// SIMATIC S7-200 project (STEP 7-Micro/WIN), CPU 224XP REL 02.01

SYMBOL_TABLE USUARIO1
P_DERECHA        I0.0
P_IZQUIERDA      I0.1
P_PARO           I0.2
R_TERMICO        I0.3
M_DERECHA        Q0.0
LED_DERECHA      Q0.1
M_IZQUIERDA      Q0.2
LED_IZQUIERDA    Q0.3
LED_PARO         Q0.4
LED_TERMICO      Q0.5
END_SYMBOL_TABLE

SYMBOL_TABLE Símbolos S7-200
Primer_ciclo_ON  SM0.1    // ON sólo en el primer ciclo
END_SYMBOL_TABLE

ORGANIZATION_BLOCK PRINCIPAL:OB1
TITLE=COMENTARIOS DEL PROGRAMA
BEGIN
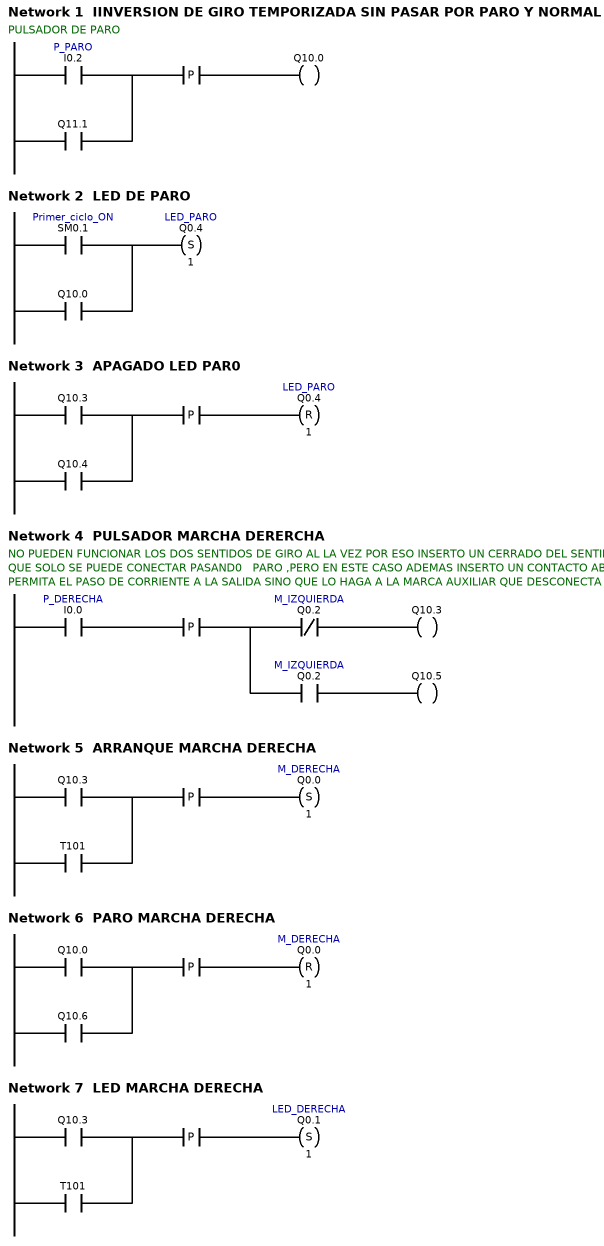
Network 1 // IINVERSION DE GIRO TEMPORIZADA SIN PASAR POR PARO Y NORMAL PASANDO POR PARO
// PULSADOR DE PARO
LD     P_PARO:I0.2
O      Q11.1
EU
=      Q10.0
Network 2 // LED DE PARO
LD     Primer_ciclo_ON:SM0.1
O      Q10.0
S      LED_PARO:Q0.4, 1
Network 3 // APAGADO LED PAR0
LD     Q10.3
O      Q10.4
EU
R      LED_PARO:Q0.4, 1
Network 4 // PULSADOR MARCHA DERERCHA
// NO PUEDEN FUNCIONAR LOS DOS SENTIDOS DE GIRO AL LA VEZ POR ESO INSERTO UN CERRADO DEL SENTIDO CONTRARIO ANTES DE LA MARCA QUE ME CONECTA AMBOS SENTIDOS DE TAL FORMA QUE SOLO SE PUEDE CONECTAR PASAND0   PARO ,PERO EN ESTE CASO ADEMAS INSERTO UN CONTACTO ABIERTO QUE CONECTA OTRA MARCA,CUAMDO YO PRESIONE EL SENTIDO QUE ELIJA NO ME PERMITA EL PASO DE CORRIENTE A LA SALIDA SINO QUE LO HAGA A LA MARCA AUXILIAR QUE DESCONECTA EL SENTIDO CONTRARIO Y TEMPORIZA PARA CONECTAR EL ELEGIDO.
LD     P_DERECHA:I0.0
EU
LPS
AN     M_IZQUIERDA:Q0.2
=      Q10.3
LPP
A      M_IZQUIERDA:Q0.2
=      Q10.5
Network 5 // ARRANQUE MARCHA DERECHA
LD     Q10.3
O      T101
EU
S      M_DERECHA:Q0.0, 1
Network 6 // PARO MARCHA DERECHA

LD     Q10.0
O      Q10.6
EU
R      M_DERECHA:Q0.0, 1
Network 7 // LED MARCHA DERECHA
LD     Q10.3
O      T101
EU
S      LED_DERECHA:Q0.1, 1
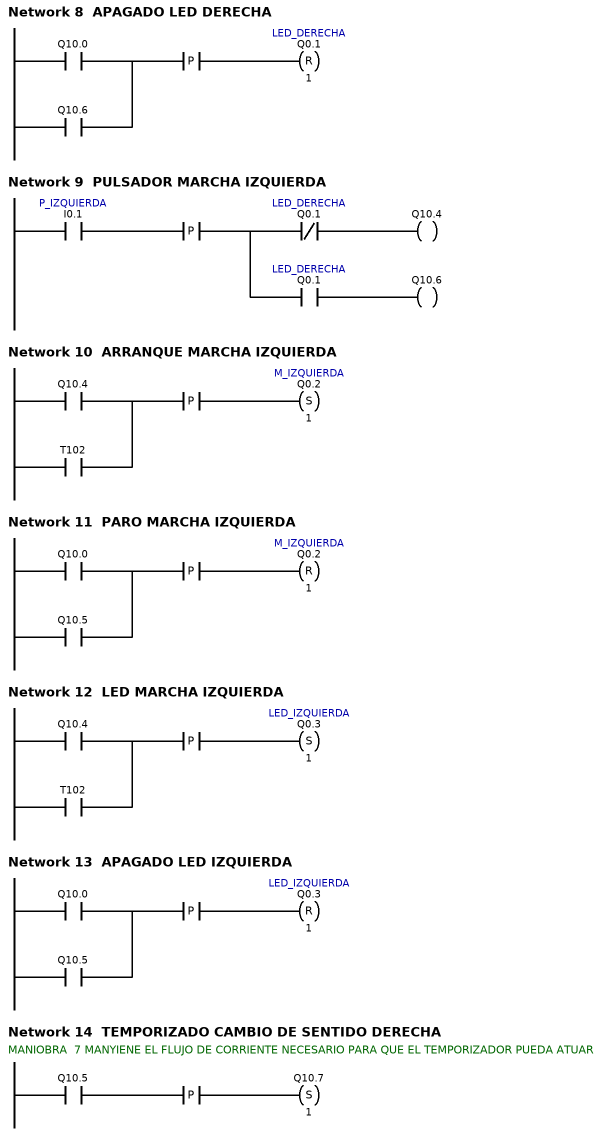
Network 8 // APAGADO LED DERECHA
LD     Q10.0
O      Q10.6
EU
R      LED_DERECHA:Q0.1, 1
Network 9 // PULSADOR MARCHA IZQUIERDA
LD     P_IZQUIERDA:I0.1
EU
LPS
AN     LED_DERECHA:Q0.1
=      Q10.4
LPP
A      LED_DERECHA:Q0.1
=      Q10.6
Network 10 // ARRANQUE MARCHA IZQUIERDA
LD     Q10.4
O      T102
EU
S      M_IZQUIERDA:Q0.2, 1
Network 11 // PARO MARCHA IZQUIERDA
LD     Q10.0
O      Q10.5
EU
R      M_IZQUIERDA:Q0.2, 1
Network 12 // LED MARCHA IZQUIERDA
LD     Q10.4
O      T102
EU
S      LED_IZQUIERDA:Q0.3, 1
Network 13 // APAGADO LED IZQUIERDA
LD     Q10.0
O      Q10.5
EU
R      LED_IZQUIERDA:Q0.3, 1
Network 14 // TEMPORIZADO CAMBIO DE SENTIDO DERECHA 
// MANIOBRA  7 MANYIENE EL FLUJO DE CORRIENTE NECESARIO PARA QUE EL TEMPORIZADOR PUEDA ATUAR 
LD     Q10.5
EU
S      Q10.7, 1
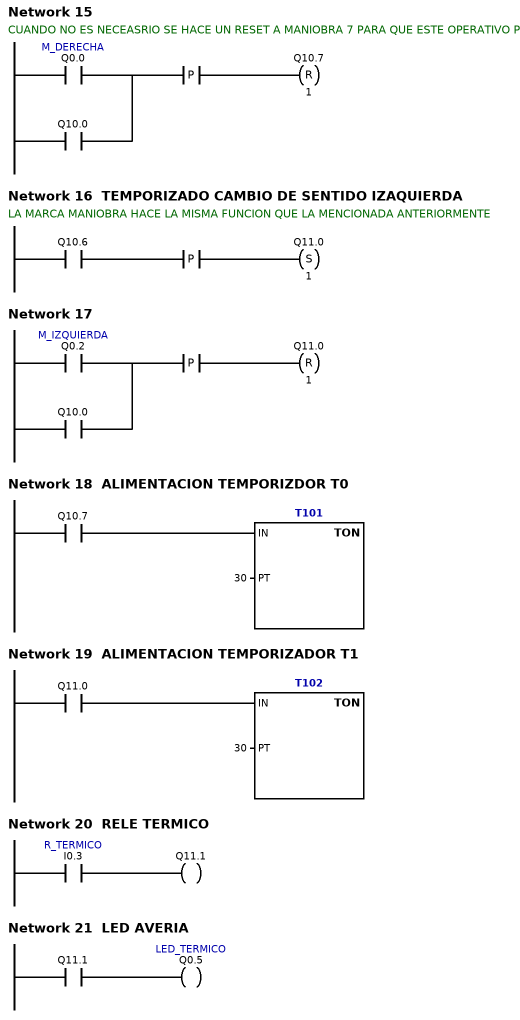
Network 15
// CUANDO NO ES NECEASRIO SE HACE UN RESET A MANIOBRA 7 PARA QUE ESTE OPERATIVO PARA LA PROXIMA VEZ QUE SEA NECESARIO.
LD     M_DERECHA:Q0.0
O      Q10.0
EU
R      Q10.7, 1
Network 16 // TEMPORIZADO CAMBIO DE SENTIDO IZAQUIERDA
// LA MARCA MANIOBRA HACE LA MISMA FUNCION QUE LA MENCIONADA ANTERIORMENTE
LD     Q10.6
EU
S      Q11.0, 1
Network 17
LD     M_IZQUIERDA:Q0.2
O      Q10.0
EU
R      Q11.0, 1
Network 18 // ALIMENTACION TEMPORIZDOR T0
LD     Q10.7
TON    T101, 30
Network 19 // ALIMENTACION TEMPORIZADOR T1
LD     Q11.0
TON    T102, 30
Network 20 // RELE TERMICO
LD     R_TERMICO:I0.3
=      Q11.1
Network 21 // LED AVERIA
LD     Q11.1
=      LED_TERMICO:Q0.5
END_ORGANIZATION_BLOCK
